FUNCTION_BLOCK ExerciseCirculationPumpsParameters
VAR_INPUT
	Interval: INT := 48; (* Central exercise interval for all damper modules (set to zero for no exercising) $(unit hour) *)
	StopVentilation: BOOL := TRUE; (* Stop ventilation during central exercise *)
	Hour: INT := 10; (* Central exercise at this hour $(unit hour) *)
	Minute: INT := 30; (* Central exercise at this minute $(unit minute) *)
	(*
	TimeChannel: TimeChannelSettings;
	StartManualExercise: BOOL;
	ExerciseStatus: BOOL;
	*)
END_VAR
VAR_OUTPUT
END_VAR
VAR
END_VAR

END_FUNCTION_BLOCK

(* stored: Version 1.1.0.1, ProductVersion 3.1.4024.6
   POU ExerciseCirculationPumpsParameters: Id {221f950b-bc06-4040-9983-aa363eb5fa79}, SpecialFunc None *)
